{attribute 'no_explicit_call' := 'do not call this function block directly'} 
// Dynamic dictionary of pointers to key and value
FUNCTION_BLOCK Dictionary EXTENDS Object IMPLEMENTS IReadOnlyDictionary
VAR_INPUT
	DefaultAllocationElemetsCount : BYTE := 10;	
END_VAR
VAR
	_ClassName : STRING := __POUNAME();

	_Array : POINTER TO GENERIC_KEY_VALUE_PAIR;
	_ArrayLength : DINT;
	_ValueCount : DINT;
END_VAR

METHOD AllocateMemory
VAR_INPUT
	elementsCount : DINT;
END_VAR
VAR
	newKeyValuePair : POINTER TO GENERIC_KEY_VALUE_PAIR;
END_VAR
newKeyValuePair := __NEW(BYTE, TO_UDINT(SIZEOF(GENERIC_KEY_VALUE_PAIR) * (_ArrayLength + elementsCount)));

IF _ValueCount > 0 THEN
	Tc2_System.MEMCPY(newKeyValuePair, _Array, TO_UDINT(SIZEOF(GENERIC_KEY_VALUE_PAIR) * _ValueCount));
END_IF
 
IF _Array <> 0 THEN
	__DELETE(_Array);
END_IF

_ArrayLength := _ArrayLength + elementsCount;

_Array := newKeyValuePair;
END_METHOD

{attribute 'monitoring' := 'call'}
PROPERTY ClassName : STRING
GET
ClassName := _ClassName;
END_GET
END_PROPERTY

METHOD Clear
VAR
	i : DINT;
END_VAR
FOR i := 0 TO _ValueCount - 1 DO
	_Array[i].Key.Release();			
	_Array[i].Value.Release();			
END_FOR	

_ValueCount := 0;
_ArrayLength := 0;

IF _Array <> 0 THEN
	__DELETE(_Array);	
END_IF
END_METHOD

METHOD ContainsGenericKey : BOOL
VAR_INPUT
	key : GENERIC_VALUE;
	releaseKey : BOOL := TRUE;
END_VAR
ContainsGenericKey := SearchKeyIndex(key.AsAnyType());

IF releaseKey THEN
	key.Release();
END_IF
END_METHOD

METHOD ContainsKey : BOOL
VAR_INPUT
	key : ANY;
END_VAR
ContainsKey := SearchKeyIndex(key);
END_METHOD

{attribute 'OPC.UA.DA.Property' := '1'}
{attribute 'monitoring' := 'call'}
PROPERTY Count : DINT
GET
Count := _ValueCount;
END_GET
END_PROPERTY

METHOD CreateEnumerator : IEnumerator
VAR
	enumerator : POINTER TO DictionaryEnumerator;
END_VAR
enumerator := __NEW(DictionaryEnumerator(dictionary := THIS^));

CreateEnumerator := enumerator^;
END_METHOD

METHOD FB_exit : BOOL
VAR_INPUT
	bInCopyCode : BOOL; // if TRUE, the exit method is called for exiting an instance that is copied afterwards (online change).
END_VAR
Clear();
END_METHOD

// Negative value returned if not found
METHOD GetGenericKeyPosition : DINT
VAR_INPUT
	key : GENERIC_VALUE;
	releaseKey : BOOL := TRUE;
END_VAR
IF NOT SearchKeyIndex(key.AsAnyType(), supposedIndex => GetGenericKeyPosition) THEN
	GetGenericKeyPosition := -1;
END_IF

IF releaseKey THEN
	key.Release();
END_IF
END_METHOD

// Negative value returned if not found
METHOD GetKeyPosition : DINT
VAR_INPUT
	key : ANY;
END_VAR
IF NOT SearchKeyIndex(key, supposedIndex => GetKeyPosition) THEN
	GetKeyPosition := -1;
END_IF
END_METHOD

METHOD GetKeyValuePairByIndex : REFERENCE TO GENERIC_KEY_VALUE_PAIR
VAR_INPUT
	index : DINT;
END_VAR
VAR
	argumentOutOfRangeException : ArgumentOutOfRangeException;
END_VAR
IF index < 0 OR_ELSE index >= _ValueCount THEN
	argumentOutOfRangeException.Throw(CurrentNamespace.Name, ClassName, __POUNAME(), __POSITION(), 'index', index);
END_IF

GetKeyValuePairByIndex REF= _Array[index];
END_METHOD

METHOD RemoveAt
VAR_INPUT
	index : DINT;
END_VAR
VAR
	argumentOutOfRangeException : ArgumentOutOfRangeException;

	i : DINT;
END_VAR
IF index < 0 OR_ELSE index >= _ValueCount THEN
	argumentOutOfRangeException.Throw(CurrentNamespace.Name, ClassName, __POUNAME(), __POSITION(), 'index', index);
END_IF

_Array[index].Key.Release();
_Array[index].Value.Release();

IF index + 2 <= _ValueCount THEN
	FOR	i := index TO _ValueCount - 2 DO
		_Array[i] := _Array[i + 1];
	END_FOR			
END_IF
	
_Array[_ValueCount - 1].Key.Reset();
_Array[_ValueCount - 1].Value.Reset();

_ValueCount := _ValueCount - 1;
END_METHOD

METHOD PROTECTED SearchKeyIndex : BOOL
VAR_INPUT
	key : __SYSTEM.AnyType;
END_VAR
VAR_OUTPUT
	supposedIndex : DINT; 
END_VAR
VAR
	lastIndex : DINT;
	minIndex : DINT;
	maxIndex : DINT;
 
	keyComparer : ByteArrayComparer;
END_VAR
IF _ValueCount = 0 THEN
	RETURN;
END_IF

lastIndex := _ValueCount - 1;
minIndex := 0;
maxIndex := lastIndex;
supposedIndex := maxIndex / 2;

WHILE minIndex <= maxIndex DO
	CASE keyComparer.Compare(_Array[supposedIndex].Key.AsAnyType(), key) OF
		// assumed key equals to seached 
		COMPARISION_RESULT.FIRST_EQUAL_TO_SECOND:
			SearchKeyIndex := TRUE;
			RETURN;

		// assumed key less than searched, move range to right
		COMPARISION_RESULT.FIRST_LESS_THAN_SECOND:
			minIndex := supposedIndex + 1;
			
		// assumed key greater than searched, move range to left	
		COMPARISION_RESULT.FIRST_GREATER_THAN_SECOND:
			maxIndex := supposedIndex - 1;
	END_CASE
	
	supposedIndex := minIndex + (maxIndex - minIndex) / 2;
END_WHILE
END_METHOD

METHOD Set : DINT
VAR_INPUT
	key : ANY;
	value : ANY;
	valueIsObject : BOOL := FALSE;
END_VAR
Set := SetGeneric(GenericValueFactory.FromAnyType(key, FALSE, TRUE), GenericValueFactory.FromAnyType(value, valueIsObject, TRUE));
END_METHOD

METHOD SetGeneric : DINT
VAR_INPUT
	key : GENERIC_VALUE;
	value : GENERIC_VALUE;
END_VAR
VAR
	genericKeyValuePair : GENERIC_KEY_VALUE_PAIR;
	index, i : DINT;
END_VAR
genericKeyValuePair.Key := key;
genericKeyValuePair.Value := value;

// if equal key found then we need to replace it
IF SearchKeyIndex(genericKeyValuePair.Key.AsAnyType(), supposedIndex => index) THEN	
	_Array[index].Key.Release(); 
	_Array[index].Value.Release(); 
ELSE
	IF _ValueCount >= _ArrayLength THEN
		AllocateMemory(DefaultAllocationElemetsCount);
	END_IF
		
	FOR i := _ValueCount - 1 TO index BY -1 DO	
		_Array[i + 1] := _Array[i];
	END_FOR

	_ValueCount := _ValueCount + 1;
END_IF

_Array[index] := genericKeyValuePair;

SetGeneric := index;
END_METHOD

{attribute 'monitoring' := 'call'}
PROPERTY Size : ULINT
GET
Size := XSIZEOF(THIS^);
END_GET
END_PROPERTY

METHOD TryGetValueByKey : BOOL
VAR_INPUT
	key : ANY;
END_VAR
VAR_OUTPUT
	value : GENERIC_VALUE;
END_VAR
VAR
	index : DINT; 
END_VAR
TryGetValueByKey := SearchKeyIndex(key, supposedIndex => index);

IF TryGetValueByKey THEN
	 value := _Array[index].Value;
END_IF
END_METHOD

METHOD TryRemove : BOOL
VAR_INPUT
	key : ANY;
END_VAR
VAR
	index : DINT;
END_VAR
TryRemove := SearchKeyIndex(key, supposedIndex => index);
 
IF TryRemove THEN
	RemoveAt(index);
END_IF
END_METHOD

END_FUNCTION_BLOCK

(* stored: Version 1.1.0.1
   POU Dictionary: Id {aa9d18ee-85a8-44b9-8978-597d9cf8b178}, SpecialFunc None
   Folder Serviceme mebers: Id {e2c68c01-e8ea-425f-ba6b-6175fdff734e}
   Method AllocateMemory: Id {0e7f768a-1410-4b70-bf65-58b5d6436902}
   Property ClassName: Id {2ba03c75-6849-4d3f-be0a-7ec3bb3723e7}
   Get Get: Id {16dbbed6-7d92-472a-aa65-fa307ed9f2d6}
   Method Clear: Id {6bbda434-8ecb-447c-84e2-06549ff7293c}
   Method ContainsGenericKey: Id {40e3952b-e79c-43eb-86c3-ebc7badec7a9}
   Method ContainsKey: Id {59c7babd-f6ce-449c-a373-7928830c9806}
   Property Count: Id {ccfee7c1-4417-440d-a786-d1356b8baab2}
   Get Get: Id {f9766b78-b24d-4be8-b437-f12592493950}
   Method CreateEnumerator: Id {5e86c797-07a7-40e5-a54a-edd93009219c}
   Method FB_exit: Id {bab70cb4-1255-41fe-9739-25af7a0667fe}
   Method GetGenericKeyPosition: Id {fbc764d5-47dd-4dd0-9946-aee3ff7c213c}
   Method GetKeyPosition: Id {bf8491de-1d63-4391-a1d1-4fca0379c7f2}
   Method GetKeyValuePairByIndex: Id {0291fd9f-109a-4434-bc5f-58af2ff03ea5}
   Method RemoveAt: Id {6ffe1d1b-7166-4447-9a30-c1b0e902f1f1}
   Method SearchKeyIndex: Id {0002c577-30ed-4f40-b96a-46bdc85d8d43}
   Method Set: Id {de4fc0d3-020e-46c6-9a06-31b5ceb0b6d1}
   Method SetGeneric: Id {94cffa05-38c9-49b3-9002-78aa4f07bd4c}
   Property Size: Id {2f97742f-3611-48c7-bd16-2c4c86e43b99}
   Get Get: Id {6d517caa-0175-488d-870c-e5bd38c78f1e}
   Method TryGetValueByKey: Id {b4d9a44b-a711-4e6d-854a-ec939d35bf59}
   Method TryRemove: Id {26dd05f9-9b20-404d-aa51-3d260ab46bbe} *)
